// TIA Portal V16 export
// export: Created 2023-03-29T11:03:45.3573179Z, ExportSetting WithDefaults, DisplayName Totally Integrated Automation Portal, DisplayVersion V16 Update 6, DisplayName TIA Portal Version Control Interface, DisplayVersion V16 Update 2, DisplayName TIA Portal Openness, DisplayVersion V16 Update 6, DisplayName STEP 7 Professional, DisplayVersion V16 Update 6, DisplayName STEP 7 Safety, DisplayVersion V16, DisplayName WinCC Advanced, DisplayVersion V16 Update 6
VAR_GLOBAL   // PLC tag table "Z9"
   isGotowość_Z_9 AT %M70.0 : Bool;   // bit gotowości wspólny
   inputAumaawariaZ_9 AT %M71.1 : Bool;   // znacznik wejście
   Hbit_REN_Z9 AT %M26.2 : Bool;
   CMD_Close_Z_9 AT %M71.6 : Bool;   // załącz zamykanie
   inputZamkniętaZ_9 AT %M70.3 : Bool;   // znacznik wejście
   inputAumaautomatZ_9 AT %M70.7 : Bool;   // znacznik wejście
   inputAumagotowośćZ_9 AT %M71.0 : Bool;   // znacznik wejście
   Hbit_Otwórz_Z9 AT %M26.4 : Bool;
   setAlarm_Moment_Z_9 AT %M71.4 : Bool;   // znacznik alarmu od momentówki w trybie zdalnym (aut/mamnual)
   Hbit_Reset_Z9 AT %M26.6 : Bool;
   Hbit_Zamknieta_Z9 AT %M26.3 : Bool;
   Hbit_Auto_Manu_Z9 AT %M26.7 : Bool;
   Byte_Status_Z9 AT %MW26 : Word;   // Słowo statusu napędu
   inputAwariaMomentZ_9 AT %M70.5 : Bool;   // znacznik wejście
   CMD_Awaria_Z_9 AT %M71.7 : Bool;   // Awaria zbiorcza
   CMD_Open_Z_9 AT %M71.5 : Bool;   // załącz otwieranie
   Hbit_Zamknij_Z9 AT %M26.5 : Bool;
   isAUMA_Z_9 AT %M52.1 : Bool;   // przęłącznik wymiany na AUMA
   Hbit_Alarm_Z9 AT %M26.0 : Bool;
   inputOtwartaZ_9 AT %M70.2 : Bool;   // znacznik wejście
   setSVMC_Z_9 AT %M71.3 : Bool;   // Znacznik polecenia zamknij w trybie automat
   inputRuch_Z_9 AT %M70.4 : Bool;
   Hbit_Otwarta_Z9 AT %M26.1 : Bool;
   inputREMT_Z_9 AT %M70.1 : Bool;   // znacznik wejście zdalne
   inputAumalokalneZ_9 AT %M70.6 : Bool;   // znacznik wejście
   setSVMO_Z_9 AT %M71.2 : Bool;   // Znacznik polecenia otwórz w trybie automat
END_VAR
